// TIA Portal project "LQG PLC TIA PORTAL" (V16)
// Vorlageprojekt für das Buch mit Zielsystem S7-1200

(* hardware
DEVICE "S7-1200-Station_1"  S7-1200 Station
   slot 0: "Baugruppenträger_0"  Rack  V1.0
   slot 1: "PLC_1"  CPU 1214C DC/DC/DC  6ES7 214-1AG40-0XB0  V4.1
   slot 3: "AQ 1x12BIT_1"  AQ1 signal board  6ES7 232-4HA30-0XB0  V1.0
DEVICE "HMI_1"  TP900 Comfort
   slot 0: "HMI_1"  TP900 Comfort  6AV2 124-0JC01-0AX0  16.0.0.0
   slot 1: "HMI_RT_1"  TP900 Comfort  6AV2 124-0JC01-0AX0  16.0.0.0
   slot 5: "HMI_1.IE_CP_1"  PROFINET Interface  16.0.0.0
      slot 1: "Interfaz PROFINET_1"  PROFINET Interface
         slot 1: "Port_1"  Port
         slot 2: "Port_2"  Port
   slot 7: "HMI_1.MPI/DP_CP_1"  MPI/DP Interface  16.0.0.0
*)

// ===== PLC "PLC_1"  CPU 1214C DC/DC/DC =====

VAR_GLOBAL   // PLC tag table "Standard-Variablentabelle"
   "L2" AT %MD40 : Real;   // entrada L1
   "L1" AT %MD44 : Real;   // entrada L2
   "Kr1" AT %MD0 : Real;   // K constant
   "Kr2" AT %MD4 : Real;   // k constant
   "L1e" AT %MD8 : Real;   // Set Point L1e
   "L2e" AT %MD12 : Real;   // Set Point L2e
   "Veq" AT %MD16 : Real;   // Set Point Veq
   "e_u" AT %MD36 : Real;   // Error del voltage
   "u_out" AT %MD48 : Real;   // Saturacion
   "v1" AT %QD4 : Real;   // sistema simulacion
   "AI_L1" AT %ID4 : Real;   // l1 de 0 a 10
   "AI_L2" AT %ID8 : Real;   // l2 de 0 a 10
   "Vp" AT %QD0 : Real;   // Salida de Control
   "FLOWMETER1" AT %ID12 : Real;
   "FLOWMETER2" AT %ID16 : Real;
   "DISCHARGE1" AT %QD8 : Real;
   "DISCHARGE2" AT %QD12 : Real;
   "hat_e1" AT %MD52 : Real;
   "hat_e2" AT %MD56 : Real;
   "Kf1_1" AT %MD60 : Real;   // Kf
   "Kf1_2" AT %MD64 : Real;   // Kf
   "Kf2_1" AT %MD68 : Real;   // Kf
   "Kf2_2" AT %MD72 : Real;   // Kf
   "e1" AT %MD76 : Real;   // error 1
   "e2" AT %MD80 : Real;   // error 2
   "dot_hat_e1" AT %MD92 : Real;   // primera derivada del error estimado 1
   "dot_hat_e2" AT %MD96 : Real;   // primera derivada del error estimado 1
   "A11" AT %MD100 : Real;
   "A12" AT %MD104 : Real;
   "A21" AT %MD108 : Real;
   "A22" AT %MD112 : Real;
   "B1" AT %MD116 : Real;
   "B2" AT %MD120 : Real;
   "resid1" AT %MD124 : Real;
   "resid2" AT %MD128 : Real;
   "pred1" AT %MD132 : Real;
   "pred2" AT %MD136 : Real;
   "corr_term1" AT %MD140 : Real;
   "corr_term2" AT %MD144 : Real;
   "disp" AT %QD16 : Real;
   "err1" AT %MD148 : Real;
   "err2" AT %MD152 : Real;
   "start" AT %I30.0 : Bool;
   "lqg11" AT %Q62.0 : Bool;
   "lqg22" AT %Q62.1 : Bool;
   "statSeed" AT %MD156 : DInt;
   "noise1" AT %MD160 : Real;
   "noise2" AT %MD164 : Real;
   "l1_ruido" AT %MD168 : Real;
   "l2_ruido" AT %MD172 : Real;
END_VAR

DATA_BLOCK "I"   // DB6
{ S7_Optimized_Access := 'TRUE' }
VERSION : 0.1
// stored: InstanceOfName lqg1
"lqg1"
BEGIN
END_DATA_BLOCK

FUNCTION_BLOCK "lqg1"   // FB2, SCL
{ S7_Optimized_Access := 'TRUE' }
VERSION : 0.1
BEGIN
   "DISCHARGE1" := 4.5;
   "DISCHARGE2" := 5;
   "v1" := 4.073 * SQRT("L2");
   "L1" := "AI_L1" * 0.3;
   "L2" := "AI_L2" * 0.3;

   "A11" := -0.010796;
   "A12" := 0.0132014;
   "A21" := 0.0;
   "A22" := -0.01320;

   "B1" := 0.000132;
   "B2" := 0.397754;

   "Kr1" := 5.938744222414906;
   "Kr2" := 3.286397049941680;

   "L1e" := 1.5000;
   "L2e" := 1.2278;


   "Veq" :=  4.5329;

   // 2) MATRIZ L DEL KALMAN

   "Kf1_1" := 0.61;
   "Kf1_2" := 0.0001;
   "Kf2_1" := 0.0001;
   "Kf2_2" := 0.61;

   // 3) CÁLCULOS PREVIOS

   "e1" := "L1" - "L1e";
   "e2" := "L2" - "L2e";


   // Cálculo del Control LQR 

   "e_u" := - ("Kr1" * "hat_e1" + "Kr2" * "hat_e2");


   // CÁLCULO DE LA DERIVADA (corr = Ax + Bu + L*error)
   "dot_hat_e1" := ("A11" * "hat_e1") + ("A12" * "hat_e2")
   + ("B1" * "e_u")
   + ("Kf1_1" * ("e1" - "hat_e1")) + ("Kf1_2" * ("e2" - "hat_e2"));

   "dot_hat_e2" := ("A21" * "hat_e1") + ("A22" * "hat_e2")
   + ("B2" * "e_u")
   + ("Kf2_1" * ("e1" - "hat_e1")) + ("Kf2_2" * ("e2" - "hat_e2"));

   // INTEGRACIÓN (Típicamente cada 50ms)
   "hat_e1" := "hat_e1" + 0.1 * "dot_hat_e1";
   "hat_e2" := "hat_e2" + 0.1 * "dot_hat_e2";

   // Visualización para debug
   "disp" := "L1";


   // 5) SEÑAL TOTAL Y SATURACIÓN


   "u_out" := "Veq" + "e_u";

   IF "u_out" > 10.0 THEN
       "u_out" := 10.0;
   ELSIF "u_out" < 0 THEN
       "u_out" := 0 ;
   END_IF;

   // 7) SALIDA AL ACTUADOR

   "Vp" :="u_out" ;
END_FUNCTION_BLOCK

FUNCTION "MHJ-PLC-Lab-Function-S71200" : Void   // FC9000, SCL
{ S7_Optimized_Access := 'TRUE' }
VERSION : 0.1
   VAR_TEMP
      rdTimeReturn : Int;
      outputTime : DTL;
      SyncVal : Byte;
      forVal : Int;
      forVal_2 : Int;
      Value : Byte;
   END_VAR
   VAR CONSTANT
      CompVal : Byte := 16#34;
      Value_01 : Byte := 16#11;
      Value_01_DW : DWord := 16#A165_D992;
      Value_02_DW : DWord := 16#58BE_4401;
   END_VAR
BEGIN

   #Value:=PEEK(area := 16#82,
        dbNumber := 0,
        byteOffset := 511);
   #Value := #Value + 1;

   POKE(area := 16#82,
        dbNumber := 0,
        byteOffset := 511,
        value := #Value);

   POKE(area:=16#81,
        dbNumber:=0,
        byteOffset:=1016,
        value:=#Value_01_DW);
   POKE(area := 16#81,
        dbNumber := 0,
        byteOffset := 1020,
        value := #Value_02_DW);

   POKE(area := 16#81,
        dbNumber := 0,
        byteOffset := 511,
        value := B#16#00);

   FOR #forVal := 0 TO 120 DO
       FOR #forVal_2:=0 TO 10 DO
           #rdTimeReturn:=RD_SYS_T(#outputTime);
           #rdTimeReturn := WR_SYS_T(#outputTime);
           #rdTimeReturn := RD_SYS_T(#outputTime);
           #rdTimeReturn := WR_SYS_T(#outputTime);
       END_FOR;
       #SyncVal:= PEEK(area := 16#81,
                      dbNumber := 0,
                      byteOffset := 511);
       IF #SyncVal = #CompVal THEN
          GOTO M_1;
       END_IF;
   END_FOR;
   RETURN;

   M_1:
   POKE(area := 16#81,
        dbNumber := 0,
        byteOffset := 511,
        value := B#16#0);
END_FUNCTION

ORGANIZATION_BLOCK "Main"   // OB1, LAD, ProgramCycle
TITLE = "Main Program Sweep (Cycle)"
{ S7_Optimized_Access := 'TRUE' }
VERSION : 0.1
   VAR_INPUT
      Initial_Call : Bool;   // Initial call of this OB
      Remanence : Bool;   // =True, if remanent data are available
   END_VAR
BEGIN

REGION Network 1: Konnektierungsbaustein für PLC-Lab
   // Im Netzwerk 1 wird der Konnektierungsbaustein für PLC-Lab aufgerufen.
   // Dieser Aufruf darf nicht entfernt werden!
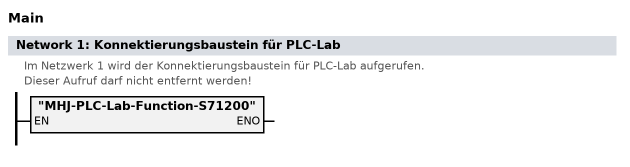
   RUNG wire#powerrail
      "MHJ-PLC-Lab-Function-S71200"()
   END_RUNG
   // the same network as SCL:
   "MHJ-PLC-Lab-Function-S71200"();
END_REGION
END_ORGANIZATION_BLOCK

ORGANIZATION_BLOCK "Cyclic interrupt"   // OB30, LAD, CyclicInterrupt
{ S7_Optimized_Access := 'TRUE' }
VERSION : 0.1
   VAR_INPUT
      Initial_Call : Bool;   // Initial call of this OB
      Event_Count : Int;   // Events discarded
   END_VAR
BEGIN

REGION Network 1
   // controller LQG
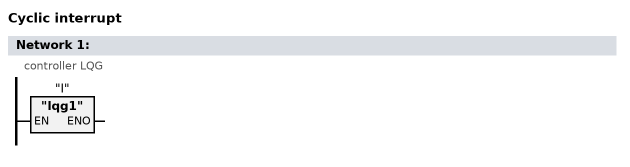
   RUNG wire#powerrail
      "I"()
   END_RUNG
   // the same network as SCL:
   "I"();   // "lqg1"
END_REGION
END_ORGANIZATION_BLOCK

(* ===== HMI "HMI_RT_1" =====
system functions are stored by id; their names below are inferred from use
connection "HMI_Conexión_1": ETHERNET, S7_1200_OMS

HMI tags "Tabla de variables estándar"
   "Número_imagen_variable" : UInt, internal
   "l1" : Real = PLC L1 AT %MD44, 1 s
   "l2" : Real = PLC L2 AT %MD40, 1 s
   "AO_u" : Real = PLC Vp AT %QD0, 1 s

screen "Imagen raíz" 800x420, template "Plantilla_1"
   on GenerateScreen: SetTag("Número_imagen_variable", 1)
   TrendView "Visor de curvas_1" at 8,5 size 787x351

Template "Plantilla_1" 800x420
   Button "Exit" at 720,360 size 78x58; TextOff 'Exit'; PictureOff "ExitRuntime_TP900_Comfort_TR"; PictureOn "ExitRuntime_TP900_Comfort_TR"
      on Release: StopRuntime(0)
   Button "Template_Button" at 640,360 size 78x58; TextOff 'Text'
   Button "Template_Button_1" at 560,360 size 78x58; TextOff 'Text'
   Button "Template_Button_2" at 480,360 size 78x58; TextOff 'Text'
   Button "Template_Button_3" at 400,360 size 78x58; TextOff 'Text'
   Button "Template_Button_4" at 321,360 size 78x58; TextOff 'Text'
   Button "Template_Button_5" at 241,360 size 78x58; TextOff 'Text'
   Button "Template_Button_6" at 161,360 size 78x58; TextOff 'Text'
   Button "Template_Button_7" at 81,360 size 78x58; TextOff 'Text'
   Button "Start screen" at 1,360 size 78x58; TextOff 'Start screen'; PictureOff "NavigateHome_TP900_Comfort_TR"; PictureOn "NavigateHome_TP900_Comfort_TR"
      on Release: ActivateScreen("Imagen raíz", 0)
*)